TYPE E_Destination :
(
	StackerA,
	StackerB,
	StackerC,
	Garbage,
	MAX_E_Destination
);
END_TYPE

(* stored: Version 1.1.0.1, ProductVersion 3.1.0.26
   DUT E_Destination: Id {3bd4f2e2-1941-46c9-ab11-2e6ce8a8a228} *)
